(* IEC 61131-3 sources: SIMERLIFT/logiwork_simerlift_80v/logiwork_simerlift_80v/HEMAbattery/src_FBD/BCU/CAN/HVCU, 4 files *)

(* ---- HVCU_Charge.iecfbd ---- *)
FUNCTION_BLOCK HVCU_Charge
  {
    Charge_Target_Current {index := 0};
    Charge_Target_Voltage {index := 1};
    Charge_Max_Current {index := 2};
    Charge_Max_Voltage {index := 3};
    CAN_Error {loc := "right", index := 5};
    CAN_CH {index := 0};
    CAN_ID {index := 1};
    width := 500;
    bgColor := "cornflowerblue";
    height := 118;
  }

  VAR
    CANRECV1 : CANRECV;
    RBITS1 : RBITS;
    RBITS2 : RBITS;
    RBITS3 : RBITS;
    RBITS4 : RBITS;
  END_VAR
  VAR_INPUT
    CAN_ID : UDINT := 0;
    CAN_CH : UDINT := 0;
  END_VAR
  VAR_OUTPUT
    Charge_Target_Current : UINT := 0;
    Charge_Target_Voltage : UINT := 0;
    Charge_Max_Current : UINT := 0;
    Charge_Max_Voltage : UINT := 0;
    CAN_Error : BOOL := 0;
  END_VAR

  (*

    // Network 1:
    NE(IN1 := CAN_ID, IN2 := 0, NE => @C(64).NE);
    CANRECV1(CH := CAN_CH, ID := CAN_ID, FMT := CAN_FORMAT#EXTENDED, PER := T#100ms, ENB := @C(64).NE);
    RBITS1(start := 0, len := 16, in := CANRECV1.DATA);
    TO_UINT(IN := RBITS1.out, TO_UINT => Charge_Target_Current);
    RBITS2(start := 16, len := 16, in := CANRECV1.DATA);
    TO_UINT(IN := RBITS2.out, TO_UINT => Charge_Target_Voltage);
    NE(IN1 := CANRECV1.RC, IN2 := 0, NE => CAN_Error);
    RBITS3(start := 32, len := 16, in := CANRECV1.DATA);
    TO_UINT(IN := RBITS3.out, TO_UINT => Charge_Max_Current);
    RBITS4(start := 48, len := 16, in := CANRECV1.DATA);
    TO_UINT(IN := RBITS4.out, TO_UINT => Charge_Max_Voltage);

  *)

  @C(64) : @F(NE), @R(340.0, 200.0, 40.0, 38.0), UDINT, @I(@N(IN1), @L(9.5)), @I(@N(IN2), @L(29.5)), @O(@N(NE), @R(9.5));
  @C(1) : @FB(CANRECV1), @R(420.0, 120.0, 120.0, 98.0), @I(@N(CH), @L(9.5)), @I(@N(ID), @L(29.5)), @I(@N(FMT), @L(49.5)), @I(@N(PER), @L(69.5)), @I(@N(ENB), @L(89.5)), @O(@N(CRX), @R(9.5)), @O(@N(DATA), @R(29.5)), @O(@N(DLC), @R(49.5)), @O(@N(MPER), @R(69.5)), @O(@N(RC), @R(89.5));
  @C(9) : @FB(RBITS1), @R(1000.0, 100.0, 120.0, 58.0), @I(@N(start), @L(9.5)), @I(@N(len), @L(29.5)), @I(@N(in), @L(49.5)), @O(@N(out), @R(9.5));
  @C(10) : @FB(RBITS2), @R(1000.0, 160.0, 120.0, 58.0), @I(@N(start), @L(9.5)), @I(@N(len), @L(29.5)), @I(@N(in), @L(49.5)), @O(@N(out), @R(9.5));
  @C(21) : @FB(RBITS3), @R(1000.0, 220.0, 120.0, 58.0), @I(@N(start), @L(9.5)), @I(@N(len), @L(29.5)), @I(@N(in), @L(49.5)), @O(@N(out), @R(9.5));
  @C(23) : @FB(RBITS4), @R(1000.0, 280.0, 120.0, 58.0), @I(@N(start), @L(9.5)), @I(@N(len), @L(29.5)), @I(@N(in), @L(49.5)), @O(@N(out), @R(9.5));
  @VF(18) : @E(T#100ms), @R(150.0, 180.0, 110.0, 19.0);
  @VF(20) : @E(CAN_FORMAT#EXTENDED), @R(40.0, 160.0, 220.0, 19.0);
  @VF(58) : @E(CAN_ID), @R(40.0, 140.0, 220.0, 19.0);
  @VF(66) : @E(0), @R(150.0, 220.0, 110.0, 19.0), UDINT;
  @VF(15) : @E(16), @R(850.0, 160.0, 110.0, 19.0), UINT;
  @VF(16) : @E(16), @R(850.0, 180.0, 110.0, 19.0), UINT;
  @VF(25) : @E(16), @R(850.0, 240.0, 110.0, 19.0), UINT;
  @VF(24) : @E(32), @R(850.0, 220.0, 110.0, 19.0), UINT;
  @VF(29) : @E(16), @R(850.0, 120.0, 110.0, 19.0), UINT;
  @VF(30) : @E(0), @R(850.0, 100.0, 110.0, 19.0), UINT;
  @VF(26) : @E(48), @R(850.0, 280.0, 110.0, 19.0), UINT;
  @VF(27) : @E(16), @R(850.0, 300.0, 110.0, 19.0), UINT;
  @VF(42) : @E(Charge_Target_Current), @R(1320.0, 100.0, 220.0, 19.0);
  @VF(43) : @E(Charge_Target_Voltage), @R(1320.0, 160.0, 220.0, 19.0);
  @VF(44) : @E(Charge_Max_Current), @R(1320.0, 220.0, 220.0, 19.0);
  @VF(45) : @E(Charge_Max_Voltage), @R(1320.0, 280.0, 220.0, 19.0);
  @C(34) : @F(TO_UINT), @R(1160.0, 280.0, 120.0, 18.0), LWORD, @I(@N(IN), @L(9.5)), @O(@N(TO_UINT), @R(9.5));
  @C(35) : @F(TO_UINT), @R(1160.0, 220.0, 120.0, 18.0), LWORD, @I(@N(IN), @L(9.5)), @O(@N(TO_UINT), @R(9.5));
  @C(36) : @F(TO_UINT), @R(1160.0, 160.0, 120.0, 18.0), LWORD, @I(@N(IN), @L(9.5)), @O(@N(TO_UINT), @R(9.5));
  @C(37) : @F(TO_UINT), @R(1160.0, 100.0, 120.0, 18.0), LWORD, @I(@N(IN), @L(9.5)), @O(@N(TO_UINT), @R(9.5));
  @VF(71) : @E(CAN_Error), @R(660.0, 200.0, 110.0, 19.0);
  @VF(69) : @E(0), @R(430.0, 220.0, 110.0, 19.0), UINT;
  @VF(22) : @E(CAN_CH), @R(40.0, 120.0, 220.0, 19.0);
  @C(51) : @F(NE), @R(580.0, 200.0, 40.0, 38.0), UINT, @I(@N(IN1), @L(9.5)), @I(@N(IN2), @L(29.5)), @O(@N(NE), @R(9.5));
  @CP(8) : 299.5, 149.5;
  @CP(12) : 809.5, 149.5;
  @CP(55) : 809.5, 209.5;
  @CP(59) : 809.5, 269.5;

  @G(6) :
     @L(@VF(58).o, @CP(8)),
     @L(@CP(8), @C(1).ID),
     @L(@CP(8), @C(64).IN1)
    ;
  @G(2) :
     @L(@VF(66).o, @C(64).IN2)
    ;
  @G(3) :
     @L(@VF(18).o, @C(1).PER)
    ;
  @G(4) :
     @L(@C(64).NE, @C(1).ENB)
    ;
  @G(5) :
     @L(@VF(20).o, @C(1).FMT)
    ;
  @G(11) :
     @L(@C(1).DATA, @CP(12)),
     @L(@CP(12), @C(9).in),
     @L(@CP(12), @CP(55)),
     @L(@CP(55), @C(10).in),
     @L(@CP(55), @CP(59)),
     @L(@CP(59), @C(21).in),
     @L(@CP(59), @C(23).in)
    ;
  @G(13) :
     @L(@VF(30).o, @C(9).start)
    ;
  @G(14) :
     @L(@VF(29).o, @C(9).len)
    ;
  @G(17) :
     @L(@VF(15).o, @C(10).start)
    ;
  @G(19) :
     @L(@VF(16).o, @C(10).len)
    ;
  @G(28) :
     @L(@VF(24).o, @C(21).start)
    ;
  @G(31) :
     @L(@VF(25).o, @C(21).len)
    ;
  @G(32) :
     @L(@VF(26).o, @C(23).start)
    ;
  @G(33) :
     @L(@VF(27).o, @C(23).len)
    ;
  @G(38) :
     @L(@C(9).out, @C(37).IN)
    ;
  @G(39) :
     @L(@C(37).TO_UINT, @VF(42).i)
    ;
  @G(40) :
     @L(@C(10).out, @C(36).IN)
    ;
  @G(41) :
     @L(@C(36).TO_UINT, @VF(43).i)
    ;
  @G(46) :
     @L(@C(21).out, @C(35).IN)
    ;
  @G(47) :
     @L(@C(35).TO_UINT, @VF(44).i)
    ;
  @G(48) :
     @L(@C(23).out, @C(34).IN)
    ;
  @G(49) :
     @L(@C(34).TO_UINT, @VF(45).i)
    ;
  @G(7) :
     @L(@VF(22).o, @C(1).CH)
    ;
  @G(50) :
     @L(@C(1).RC, @C(51).IN1)
    ;
  @G(52) :
     @L(@C(51).NE, @VF(71).i)
    ;
  @G(53) :
     @L(@VF(69).o, @C(51).IN2)
    ;
END_FUNCTION_BLOCK

(* ---- HVCU_Config.iecfbd ---- *)
FUNCTION_BLOCK HVCU_Config
  {
    CAN_CH {index := 0};
    CAN_ID {index := 1};
    cmd0 {index := 0};
    CAN_Error {index := 4};
    width := 500;
    height := 98;
    bgColor := "cornflowerblue";
  }

  VAR
    CANRECV1 : CANRECV;
  END_VAR
  VAR_INPUT
    CAN_CH : UDINT := 0;
    CAN_ID : UDINT := 0;
  END_VAR
  VAR_OUTPUT
    cmd0 : USINT := 0;
    CAN_Error : BOOL;
    cmd1 : USINT;
    cmd2 : USINT;
    cmd3 : USINT;
  END_VAR

  (*

    // Network 1:
    NE(IN1 := CAN_ID, IN2 := 0, NE => @C(64).NE);
    CANRECV1(CH := CAN_CH, ID := CAN_ID, FMT := CAN_FORMAT#EXTENDED, PER := T#3000ms, ENB := @C(64).NE);
    RBIT(start := 0, len := 8, INbit := CANRECV1.DATA, OUTbit => @C(24).OUTbit);
    TO_USINT(IN := @C(24).OUTbit, TO_USINT => cmd0);
    RBIT(start := 8, len := 8, INbit := CANRECV1.DATA, OUTbit => @C(35).OUTbit);
    TO_USINT(IN := @C(35).OUTbit, TO_USINT => cmd1);
    NE(IN1 := CANRECV1.RC, IN2 := 0, NE => CAN_Error);
    RBIT(start := 16, len := 8, INbit := CANRECV1.DATA, OUTbit => @C(11).OUTbit);
    TO_USINT(IN := @C(11).OUTbit, TO_USINT => cmd2);
    RBIT(start := 24, len := 8, INbit := CANRECV1.DATA, OUTbit => @C(40).OUTbit);
    TO_USINT(IN := @C(40).OUTbit, TO_USINT => cmd3);

  *)

  @C(1) : @FB(CANRECV1), @R(430.0, 100.0, 120.0, 98.0), @I(@N(CH), @L(9.5)), @I(@N(ID), @L(29.5)), @I(@N(FMT), @L(49.5)), @I(@N(PER), @L(69.5)), @I(@N(ENB), @L(89.5)), @O(@N(CRX), @R(9.5)), @O(@N(DATA), @R(29.5)), @O(@N(DLC), @R(49.5)), @O(@N(MPER), @R(69.5)), @O(@N(RC), @R(89.5));
  @C(64) : @F(NE), @R(350.0, 180.0, 40.0, 38.0), UDINT, @I(@N(IN1), @L(9.5)), @I(@N(IN2), @L(29.5)), @O(@N(NE), @R(9.5));
  @C(51) : @F(NE), @R(590.0, 180.0, 40.0, 38.0), UINT, @I(@N(IN1), @L(9.5)), @I(@N(IN2), @L(29.5)), @O(@N(NE), @R(9.5));
  @VF(20) : @E(CAN_FORMAT#EXTENDED), @R(50.0, 140.0, 220.0, 19.0);
  @VF(18) : @E(T#3000ms), @R(160.0, 160.0, 110.0, 19.0);
  @VF(66) : @E(0), @R(160.0, 200.0, 110.0, 19.0), UDINT;
  @VF(69) : @E(0), @R(440.0, 200.0, 110.0, 19.0), UINT;
  @VF(6) : @E(CAN_CH), @R(50.0, 100.0, 220.0, 19.0);
  @VF(7) : @E(CAN_ID), @R(50.0, 120.0, 220.0, 19.0);
  @VF(30) : @E(16), @R(820.0, 200.0, 110.0, 19.0), INT;
  @VF(29) : @E(8), @R(820.0, 220.0, 110.0, 19.0), INT;
  @C(11) : @F(RBIT), @R(970.0, 200.0, 120.0, 58.0), @I(@N(start), @L(9.5)), @I(@N(len), @L(29.5)), @I(@N(INbit), @L(49.5)), @O(@N(OUTbit), @R(9.5));
  @C(23) : @F(TO_USINT), @R(1130.0, 80.0, 120.0, 18.0), LWORD, @I(@N(IN), @L(9.5)), @O(@N(TO_USINT), @R(9.5));
  @C(24) : @F(RBIT), @R(970.0, 80.0, 120.0, 58.0), @I(@N(start), @L(9.5)), @I(@N(len), @L(29.5)), @I(@N(INbit), @L(49.5)), @O(@N(OUTbit), @R(9.5));
  @VF(25) : @E(0), @R(820.0, 80.0, 110.0, 19.0), INT;
  @VF(26) : @E(8), @R(820.0, 100.0, 110.0, 19.0), INT;
  @VF(27) : @E(cmd0), @R(1290.0, 80.0, 220.0, 19.0);
  @C(35) : @F(RBIT), @R(970.0, 140.0, 120.0, 58.0), @I(@N(start), @L(9.5)), @I(@N(len), @L(29.5)), @I(@N(INbit), @L(49.5)), @O(@N(OUTbit), @R(9.5));
  @VF(36) : @E(8), @R(820.0, 140.0, 110.0, 19.0), INT;
  @VF(37) : @E(8), @R(820.0, 160.0, 110.0, 19.0), INT;
  @VF(17) : @E(CAN_Error), @R(650.0, 180.0, 140.0, 19.0);
  @C(40) : @F(RBIT), @R(970.0, 260.0, 120.0, 58.0), @I(@N(start), @L(9.5)), @I(@N(len), @L(29.5)), @I(@N(INbit), @L(49.5)), @O(@N(OUTbit), @R(9.5));
  @VF(46) : @E(8), @R(820.0, 280.0, 110.0, 19.0), INT;
  @VF(47) : @E(24), @R(820.0, 260.0, 110.0, 19.0), INT;
  @C(12) : @F(TO_USINT), @R(1130.0, 140.0, 120.0, 18.0), LWORD, @I(@N(IN), @L(9.5)), @O(@N(TO_USINT), @R(9.5));
  @VF(15) : @E(cmd1), @R(1290.0, 140.0, 220.0, 19.0);
  @C(22) : @F(TO_USINT), @R(1130.0, 200.0, 120.0, 18.0), LWORD, @I(@N(IN), @L(9.5)), @O(@N(TO_USINT), @R(9.5));
  @VF(34) : @E(cmd2), @R(1290.0, 200.0, 220.0, 19.0);
  @C(42) : @F(TO_USINT), @R(1130.0, 260.0, 120.0, 18.0), LWORD, @I(@N(IN), @L(9.5)), @O(@N(TO_USINT), @R(9.5));
  @VF(44) : @E(cmd3), @R(1290.0, 260.0, 220.0, 19.0);
  @CP(10) : 309.5, 129.5;
  @CP(43) : 949.5, 129.5;

  @G(4) :
     @L(@C(64).NE, @C(1).ENB)
    ;
  @G(2) :
     @L(@VF(66).o, @C(64).IN2)
    ;
  @G(3) :
     @L(@VF(18).o, @C(1).PER)
    ;
  @G(5) :
     @L(@VF(20).o, @C(1).FMT)
    ;
  @G(53) :
     @L(@VF(69).o, @C(51).IN2)
    ;
  @G(50) :
     @L(@C(1).RC, @C(51).IN1)
    ;
  @G(8) :
     @L(@VF(7).o, @CP(10)),
     @L(@CP(10), @C(1).ID),
     @L(@CP(10), @C(64).IN1)
    ;
  @G(9) :
     @L(@VF(6).o, @C(1).CH)
    ;
  @G(13) :
     @L(@VF(30).o, @C(11).start)
    ;
  @G(14) :
     @L(@VF(29).o, @C(11).len)
    ;
  @G(28) :
     @L(@VF(25).o, @C(24).start)
    ;
  @G(31) :
     @L(@C(24).OUTbit, @C(23).IN)
    ;
  @G(32) :
     @L(@VF(26).o, @C(24).len)
    ;
  @G(33) :
     @L(@C(23).TO_USINT, @VF(27).i)
    ;
  @G(21) :
     @L(@C(1).DATA, @CP(43)),
     @L(@CP(43), @C(24).INbit),
     @L(@CP(43), @C(35).INbit),
     @L(@CP(43), @C(11).INbit),
     @L(@CP(43), @C(40).INbit)
    ;
  @G(39) :
     @L(@VF(36).o, @C(35).start)
    ;
  @G(41) :
     @L(@VF(37).o, @C(35).len)
    ;
  @G(19) :
     @L(@C(51).NE, @VF(17).i)
    ;
  @G(49) :
     @L(@VF(46).o, @C(40).len)
    ;
  @G(52) :
     @L(@VF(47).o, @C(40).start)
    ;
  @G(16) :
     @L(@C(12).TO_USINT, @VF(15).i)
    ;
  @G(38) :
     @L(@C(22).TO_USINT, @VF(34).i)
    ;
  @G(45) :
     @L(@C(42).TO_USINT, @VF(44).i)
    ;
  @G(48) :
     @L(@C(35).OUTbit, @C(12).IN)
    ;
  @G(54) :
     @L(@C(11).OUTbit, @C(22).IN)
    ;
  @G(55) :
     @L(@C(40).OUTbit, @C(42).IN)
    ;
END_FUNCTION_BLOCK

(* ---- HVCU_Control_State.iecfbd ---- *)
FUNCTION_BLOCK HVCU_Control_State
  {
    Battey_State_BCU_00 {index := 0};
    Battey_State_BCU_01 {index := 1};
    Battey_State_BCU_02 {index := 2};
    Battey_State_BCU_03 {index := 3};
    CAN_CH {index := 0};
    CAN_ID {index := 1};
    width := 500;
    height := 198;
    bgColor := "cornflowerblue";
  }

  VAR
    CANRECV1 : CANRECV;
  END_VAR
  VAR_INPUT
    CAN_ID : UDINT := 0;
    CAN_CH : UDINT := 0;
  END_VAR
  VAR_OUTPUT
    Battey_State_BCU_00 : USINT := 0;
    Battey_State_BCU_01 : USINT := 0;
    Battey_State_BCU_02 : USINT := 0;
    Battey_State_BCU_03 : USINT := 0;
    IMDCtrl_BCU0 : BOOL;
    CAN_Error : BOOL;
  END_VAR

  (*

    // Network 1:
    NE(IN1 := CAN_ID, IN2 := 0, NE => @C(64).NE);
    CANRECV1(CH := CAN_CH, ID := CAN_ID, FMT := CAN_FORMAT#EXTENDED, PER := T#2s, ENB := @C(64).NE);
    RBIT(start := 0, len := 8, INbit := CANRECV1.DATA, OUTbit => @C(9).OUTbit);
    TO_USINT(IN := @C(9).OUTbit, TO_USINT => Battey_State_BCU_00);
    RBIT(start := 8, len := 8, INbit := CANRECV1.DATA, OUTbit => @C(10).OUTbit);
    TO_USINT(IN := @C(10).OUTbit, TO_USINT => Battey_State_BCU_01);
    NE(IN1 := CANRECV1.RC, IN2 := 0, NE => CAN_Error);
    RBIT(start := 16, len := 8, INbit := CANRECV1.DATA, OUTbit => @C(13).OUTbit);
    TO_USINT(IN := @C(13).OUTbit, TO_USINT => Battey_State_BCU_02);
    RBIT(start := 24, len := 8, INbit := CANRECV1.DATA, OUTbit => @C(14).OUTbit);
    TO_USINT(IN := @C(14).OUTbit, TO_USINT => Battey_State_BCU_03);
    RBIT(start := 32, len := 1, INbit := CANRECV1.DATA, OUTbit => @C(17).OUTbit);
    TO_BOOL(IN := @C(17).OUTbit, TO_BOOL => IMDCtrl_BCU0);

  *)

  @C(64) : @F(NE), @R(320.0, 120.0, 40.0, 38.0), UDINT, @I(@N(IN1), @L(9.5)), @I(@N(IN2), @L(29.5)), @O(@N(NE), @R(9.5));
  @C(1) : @FB(CANRECV1), @R(400.0, 40.0, 120.0, 98.0), @I(@N(CH), @L(9.5)), @I(@N(ID), @L(29.5)), @I(@N(FMT), @L(49.5)), @I(@N(PER), @L(69.5)), @I(@N(ENB), @L(89.5)), @O(@N(CRX), @R(9.5)), @O(@N(DATA), @R(29.5)), @O(@N(DLC), @R(49.5)), @O(@N(MPER), @R(69.5)), @O(@N(RC), @R(89.5));
  @C(76) : @F(TO_USINT), @R(1140.0, 80.0, 120.0, 18.0), LWORD, @I(@N(IN), @L(9.5)), @O(@N(TO_USINT), @R(9.5));
  @C(73) : @F(TO_USINT), @R(1140.0, 20.0, 120.0, 18.0), LWORD, @I(@N(IN), @L(9.5)), @O(@N(TO_USINT), @R(9.5));
  @C(92) : @F(TO_USINT), @R(1140.0, 140.0, 120.0, 18.0), LWORD, @I(@N(IN), @L(9.5)), @O(@N(TO_USINT), @R(9.5));
  @VF(18) : @E(T#2s), @R(130.0, 100.0, 110.0, 19.0);
  @VF(20) : @E(CAN_FORMAT#EXTENDED), @R(20.0, 80.0, 220.0, 19.0);
  @VF(58) : @E(CAN_ID), @R(20.0, 60.0, 220.0, 19.0);
  @VF(66) : @E(0), @R(130.0, 140.0, 110.0, 19.0), UDINT;
  @VF(115) : @E(0), @R(410.0, 140.0, 110.0, 19.0), UINT;
  @VF(15) : @E(8), @R(830.0, 80.0, 110.0, 19.0), INT;
  @VF(16) : @E(8), @R(830.0, 100.0, 110.0, 19.0), INT;
  @VF(25) : @E(8), @R(830.0, 160.0, 110.0, 19.0), INT;
  @VF(24) : @E(16), @R(830.0, 140.0, 110.0, 19.0), INT;
  @VF(27) : @E(8), @R(830.0, 220.0, 110.0, 19.0), INT;
  @VF(26) : @E(24), @R(830.0, 200.0, 110.0, 19.0), INT;
  @VF(29) : @E(8), @R(830.0, 40.0, 110.0, 19.0), INT;
  @VF(30) : @E(0), @R(830.0, 20.0, 110.0, 19.0), INT;
  @VF(36) : @E(32), @R(830.0, 260.0, 110.0, 19.0), INT;
  @VF(37) : @E(1), @R(830.0, 280.0, 110.0, 19.0), INT;
  @C(56) : @F(TO_USINT), @R(1140.0, 200.0, 120.0, 18.0), LWORD, @I(@N(IN), @L(9.5)), @O(@N(TO_USINT), @R(9.5));
  @VF(69) : @E(Battey_State_BCU_00), @R(1300.0, 20.0, 220.0, 19.0);
  @VF(70) : @E(Battey_State_BCU_01), @R(1300.0, 80.0, 220.0, 19.0);
  @VF(71) : @E(Battey_State_BCU_02), @R(1300.0, 140.0, 220.0, 19.0);
  @VF(72) : @E(Battey_State_BCU_03), @R(1300.0, 200.0, 220.0, 19.0);
  @VF(94) : @E(CAN_CH), @R(20.0, 40.0, 220.0, 19.0);
  @C(95) : @F(NE), @R(560.0, 120.0, 40.0, 38.0), UINT, @I(@N(IN1), @L(9.5)), @I(@N(IN2), @L(29.5)), @O(@N(NE), @R(9.5));
  @C(9) : @F(RBIT), @R(980.0, 20.0, 120.0, 58.0), @I(@N(start), @L(9.5)), @I(@N(len), @L(29.5)), @I(@N(INbit), @L(49.5)), @O(@N(OUTbit), @R(9.5));
  @C(10) : @F(RBIT), @R(980.0, 80.0, 120.0, 58.0), @I(@N(start), @L(9.5)), @I(@N(len), @L(29.5)), @I(@N(INbit), @L(49.5)), @O(@N(OUTbit), @R(9.5));
  @C(13) : @F(RBIT), @R(980.0, 140.0, 120.0, 58.0), @I(@N(start), @L(9.5)), @I(@N(len), @L(29.5)), @I(@N(INbit), @L(49.5)), @O(@N(OUTbit), @R(9.5));
  @C(14) : @F(RBIT), @R(980.0, 200.0, 120.0, 58.0), @I(@N(start), @L(9.5)), @I(@N(len), @L(29.5)), @I(@N(INbit), @L(49.5)), @O(@N(OUTbit), @R(9.5));
  @C(17) : @F(RBIT), @R(980.0, 260.0, 120.0, 58.0), @I(@N(start), @L(9.5)), @I(@N(len), @L(29.5)), @I(@N(INbit), @L(49.5)), @O(@N(OUTbit), @R(9.5));
  @VF(75) : @E(CAN_Error), @R(620.0, 120.0, 140.0, 19.0);
  @VF(78) : @E(IMDCtrl_BCU0), @R(1310.0, 260.0, 140.0, 19.0);
  @C(32) : @F(TO_BOOL), @R(1140.0, 260.0, 120.0, 18.0), LWORD, @I(@N(IN), @L(9.5)), @O(@N(TO_BOOL), @R(9.5));
  @CP(8) : 279.5, 69.5;
  @CP(12) : 789.5, 69.5;
  @CP(55) : 789.5, 129.5;
  @CP(59) : 789.5, 189.5;
  @CP(60) : 789.5, 249.5;

  @G(2) :
     @L(@VF(66).o, @C(64).IN2)
    ;
  @G(6) :
     @L(@VF(58).o, @CP(8)),
     @L(@CP(8), @C(1).ID),
     @L(@CP(8), @C(64).IN1)
    ;
  @G(3) :
     @L(@VF(18).o, @C(1).PER)
    ;
  @G(4) :
     @L(@C(64).NE, @C(1).ENB)
    ;
  @G(5) :
     @L(@VF(20).o, @C(1).FMT)
    ;
  @G(11) :
     @L(@C(1).DATA, @CP(12)),
     @L(@CP(12), @CP(55)),
     @L(@CP(55), @CP(59)),
     @L(@CP(59), @CP(60)),
     @L(@CP(12), @C(9).INbit),
     @L(@CP(55), @C(10).INbit),
     @L(@CP(59), @C(13).INbit),
     @L(@CP(60), @C(14).INbit),
     @L(@CP(60), @C(17).INbit)
    ;
  @G(80) :
     @L(@C(73).TO_USINT, @VF(69).i)
    ;
  @G(83) :
     @L(@C(76).TO_USINT, @VF(70).i)
    ;
  @G(84) :
     @L(@C(92).TO_USINT, @VF(71).i)
    ;
  @G(85) :
     @L(@C(56).TO_USINT, @VF(72).i)
    ;
  @G(7) :
     @L(@VF(94).o, @C(1).CH)
    ;
  @G(96) :
     @L(@C(1).RC, @C(95).IN1)
    ;
  @G(98) :
     @L(@VF(115).o, @C(95).IN2)
    ;
  @G(33) :
     @L(@C(14).OUTbit, @C(56).IN)
    ;
  @G(34) :
     @L(@C(13).OUTbit, @C(92).IN)
    ;
  @G(35) :
     @L(@C(10).OUTbit, @C(76).IN)
    ;
  @G(40) :
     @L(@C(9).OUTbit, @C(73).IN)
    ;
  @G(41) :
     @L(@VF(30).o, @C(9).start)
    ;
  @G(42) :
     @L(@VF(29).o, @C(9).len)
    ;
  @G(43) :
     @L(@VF(15).o, @C(10).start)
    ;
  @G(44) :
     @L(@VF(16).o, @C(10).len)
    ;
  @G(45) :
     @L(@VF(24).o, @C(13).start)
    ;
  @G(50) :
     @L(@VF(25).o, @C(13).len)
    ;
  @G(51) :
     @L(@VF(27).o, @C(14).len)
    ;
  @G(52) :
     @L(@VF(26).o, @C(14).start)
    ;
  @G(91) :
     @L(@VF(37).o, @C(17).len)
    ;
  @G(93) :
     @L(@VF(36).o, @C(17).start)
    ;
  @G(77) :
     @L(@C(95).NE, @VF(75).i)
    ;
  @G(54) :
     @L(@C(17).OUTbit, @C(32).IN)
    ;
  @G(79) :
     @L(@C(32).TO_BOOL, @VF(78).i)
    ;
END_FUNCTION_BLOCK

(* ---- HVCU_Power.iecfbd ---- *)
FUNCTION_BLOCK HVCU_Power
  {
    CAN_Error {loc := "right", index := 5};
    HVCU_Total_Voltage {index := 0};
    HVCU_Total_Current {index := 1};
    HVCU_Instant_Current {index := 2};
    HVCU_Available_Energy {index := 3};
    CAN_CH {index := 0};
    CAN_ID {index := 1};
    width := 500;
    bgColor := "cornflowerblue";
    height := 118;
  }

  VAR
    RBITS3 : RBITS;
    RBITS4 : RBITS;
    RBITS2 : RBITS;
    RBITS1 : RBITS;
    CANRECV1 : CANRECV;
  END_VAR
  VAR_INPUT
    CAN_ID : UDINT := 0;
    CAN_CH : UDINT := 0;
  END_VAR
  VAR_OUTPUT
    HVCU_Total_Voltage : UINT := 0;
    HVCU_Total_Current : UINT := 0;
    HVCU_Instant_Current : UINT := 0;
    HVCU_Available_Energy : UINT := 0;
    CAN_Error : BOOL := 0;
  END_VAR

  (*

    // Network 1:
    NE(IN1 := CAN_ID, IN2 := 0, NE => @C(64).NE);
    CANRECV1(CH := CAN_CH, ID := CAN_ID, FMT := CAN_FORMAT#EXTENDED, PER := T#100ms, ENB := @C(64).NE);
    RBITS1(start := 0, len := 16, in := CANRECV1.DATA);
    TO_UINT(IN := RBITS1.out, TO_UINT => HVCU_Total_Voltage);
    RBITS2(start := 16, len := 16, in := CANRECV1.DATA);
    TO_UINT(IN := RBITS2.out, TO_UINT => HVCU_Total_Current);
    NE(IN1 := CANRECV1.RC, IN2 := 0, NE => CAN_Error);
    RBITS3(start := 32, len := 16, in := CANRECV1.DATA);
    TO_UINT(IN := RBITS3.out, TO_UINT => HVCU_Instant_Current);
    RBITS4(start := 48, len := 16, in := CANRECV1.DATA);
    TO_UINT(IN := RBITS4.out, TO_UINT => HVCU_Available_Energy);

  *)

  @C(34) : @F(TO_UINT), @R(1160.0, 260.0, 120.0, 18.0), LWORD, @I(@N(IN), @L(9.5)), @O(@N(TO_UINT), @R(9.5));
  @C(35) : @F(TO_UINT), @R(1160.0, 200.0, 120.0, 18.0), LWORD, @I(@N(IN), @L(9.5)), @O(@N(TO_UINT), @R(9.5));
  @C(21) : @FB(RBITS3), @R(1000.0, 200.0, 120.0, 58.0), @I(@N(start), @L(9.5)), @I(@N(len), @L(29.5)), @I(@N(in), @L(49.5)), @O(@N(out), @R(9.5));
  @C(23) : @FB(RBITS4), @R(1000.0, 260.0, 120.0, 58.0), @I(@N(start), @L(9.5)), @I(@N(len), @L(29.5)), @I(@N(in), @L(49.5)), @O(@N(out), @R(9.5));
  @C(10) : @FB(RBITS2), @R(1000.0, 140.0, 120.0, 58.0), @I(@N(start), @L(9.5)), @I(@N(len), @L(29.5)), @I(@N(in), @L(49.5)), @O(@N(out), @R(9.5));
  @C(36) : @F(TO_UINT), @R(1160.0, 140.0, 120.0, 18.0), LWORD, @I(@N(IN), @L(9.5)), @O(@N(TO_UINT), @R(9.5));
  @C(9) : @FB(RBITS1), @R(1000.0, 80.0, 120.0, 58.0), @I(@N(start), @L(9.5)), @I(@N(len), @L(29.5)), @I(@N(in), @L(49.5)), @O(@N(out), @R(9.5));
  @C(37) : @F(TO_UINT), @R(1160.0, 80.0, 120.0, 18.0), LWORD, @I(@N(IN), @L(9.5)), @O(@N(TO_UINT), @R(9.5));
  @C(1) : @FB(CANRECV1), @R(420.0, 100.0, 120.0, 98.0), @I(@N(CH), @L(9.5)), @I(@N(ID), @L(29.5)), @I(@N(FMT), @L(49.5)), @I(@N(PER), @L(69.5)), @I(@N(ENB), @L(89.5)), @O(@N(CRX), @R(9.5)), @O(@N(DATA), @R(29.5)), @O(@N(DLC), @R(49.5)), @O(@N(MPER), @R(69.5)), @O(@N(RC), @R(89.5));
  @C(64) : @F(NE), @R(340.0, 180.0, 40.0, 38.0), UDINT, @I(@N(IN1), @L(9.5)), @I(@N(IN2), @L(29.5)), @O(@N(NE), @R(9.5));
  @VF(15) : @E(16), @R(850.0, 140.0, 110.0, 19.0), UINT;
  @VF(16) : @E(16), @R(850.0, 160.0, 110.0, 19.0), UINT;
  @VF(25) : @E(16), @R(850.0, 220.0, 110.0, 19.0), UINT;
  @VF(24) : @E(32), @R(850.0, 200.0, 110.0, 19.0), UINT;
  @VF(27) : @E(16), @R(850.0, 280.0, 110.0, 19.0), UINT;
  @VF(26) : @E(48), @R(850.0, 260.0, 110.0, 19.0), UINT;
  @VF(29) : @E(16), @R(850.0, 100.0, 110.0, 19.0), UINT;
  @VF(30) : @E(0), @R(850.0, 80.0, 110.0, 19.0), UINT;
  @VF(66) : @E(0), @R(150.0, 200.0, 110.0, 19.0), UDINT;
  @VF(18) : @E(T#100ms), @R(150.0, 160.0, 110.0, 19.0);
  @VF(20) : @E(CAN_FORMAT#EXTENDED), @R(40.0, 140.0, 220.0, 19.0);
  @VF(58) : @E(CAN_ID), @R(40.0, 120.0, 220.0, 19.0);
  @VF(39) : @E(HVCU_Total_Voltage), @R(1320.0, 80.0, 220.0, 19.0);
  @VF(41) : @E(HVCU_Total_Current), @R(1320.0, 140.0, 220.0, 19.0);
  @VF(42) : @E(HVCU_Instant_Current), @R(1320.0, 200.0, 220.0, 19.0);
  @VF(43) : @E(HVCU_Available_Energy), @R(1320.0, 260.0, 220.0, 19.0);
  @VF(71) : @E(CAN_Error), @R(660.0, 180.0, 110.0, 19.0);
  @VF(69) : @E(0), @R(430.0, 200.0, 110.0, 19.0), UINT;
  @VF(22) : @E(CAN_CH), @R(40.0, 100.0, 220.0, 19.0);
  @C(51) : @F(NE), @R(580.0, 180.0, 40.0, 38.0), UINT, @I(@N(IN1), @L(9.5)), @I(@N(IN2), @L(29.5)), @O(@N(NE), @R(9.5));
  @CP(12) : 809.5, 129.5;
  @CP(55) : 809.5, 189.5;
  @CP(59) : 809.5, 249.5;
  @CP(8) : 299.5, 129.5;

  @G(46) :
     @L(@C(21).out, @C(35).IN)
    ;
  @G(48) :
     @L(@C(23).out, @C(34).IN)
    ;
  @G(19) :
     @L(@VF(16).o, @C(10).len)
    ;
  @G(28) :
     @L(@VF(24).o, @C(21).start)
    ;
  @G(31) :
     @L(@VF(25).o, @C(21).len)
    ;
  @G(32) :
     @L(@VF(26).o, @C(23).start)
    ;
  @G(33) :
     @L(@VF(27).o, @C(23).len)
    ;
  @G(17) :
     @L(@VF(15).o, @C(10).start)
    ;
  @G(40) :
     @L(@C(10).out, @C(36).IN)
    ;
  @G(14) :
     @L(@VF(29).o, @C(9).len)
    ;
  @G(13) :
     @L(@VF(30).o, @C(9).start)
    ;
  @G(38) :
     @L(@C(9).out, @C(37).IN)
    ;
  @G(11) :
     @L(@C(1).DATA, @CP(12)),
     @L(@CP(12), @C(9).in),
     @L(@CP(12), @CP(55)),
     @L(@CP(55), @C(10).in),
     @L(@CP(55), @CP(59)),
     @L(@CP(59), @C(21).in),
     @L(@CP(59), @C(23).in)
    ;
  @G(4) :
     @L(@C(64).NE, @C(1).ENB)
    ;
  @G(6) :
     @L(@VF(58).o, @CP(8)),
     @L(@CP(8), @C(1).ID),
     @L(@CP(8), @C(64).IN1)
    ;
  @G(2) :
     @L(@VF(66).o, @C(64).IN2)
    ;
  @G(3) :
     @L(@VF(18).o, @C(1).PER)
    ;
  @G(5) :
     @L(@VF(20).o, @C(1).FMT)
    ;
  @G(44) :
     @L(@C(37).TO_UINT, @VF(39).i)
    ;
  @G(45) :
     @L(@C(36).TO_UINT, @VF(41).i)
    ;
  @G(47) :
     @L(@C(35).TO_UINT, @VF(42).i)
    ;
  @G(49) :
     @L(@C(34).TO_UINT, @VF(43).i)
    ;
  @G(7) :
     @L(@VF(22).o, @C(1).CH)
    ;
  @G(50) :
     @L(@C(1).RC, @C(51).IN1)
    ;
  @G(52) :
     @L(@C(51).NE, @VF(71).i)
    ;
  @G(53) :
     @L(@VF(69).o, @C(51).IN2)
    ;
END_FUNCTION_BLOCK
